// TIA Portal V17 export
// export: Created 2024-06-16T17:47:40.0155187Z, ExportSetting WithDefaults, DisplayName Totally Integrated Automation Portal, DisplayVersion V17, DisplayName TIA Portal Openness, DisplayVersion V17, DisplayName TIA Portal Version Control Interface, DisplayVersion V17, DisplayName STEP 7 Professional, DisplayVersion V17, DisplayName STEP 7 Safety, DisplayVersion V17, DisplayName WinCC Professional, DisplayVersion V17
VAR_GLOBAL   // PLC tag table "St4_Out"
   IO_Sortir_Loquet AT %Q2.4 : Bool;   // Sortir : Loquet (Déplacement Barquette)
   IO_Sortir_PoussoirC AT %Q2.5 : Bool;   // Sortir : Poussoir Z-OK
   IO_Ouverture_PincesC AT %Q2.6 : Bool;   // Ouverture : Pinces C
   IO_Fermeture_PincesC AT %Q2.7 : Bool;   // Fermeture : Pinces C
   IO_Vy_C AT %Q3.0 : Bool;   // Zone Conforme pleine - A vidanger
   IO_Sortir_PoussoirNC AT %Q3.1 : Bool;   // Sortir Poussoir NC
   IO_Ouverture_PincesNC AT %Q3.2 : Bool;   // Ouverture Pinces NC
   IO_Fermeture_PincesNC AT %Q3.3 : Bool;   // Fermeture Pinces NC
   IO_Vy_NC AT %Q3.4 : Bool;   // Zone Non-Conforme pleine - A vidanger
END_VAR
